(*
SPDX-FileCopyrightText: Â© 2026 Oleksandr Tiutyk <trofimich@gmail.com>
SPDX-License-Identifier: MIT
License: https://opensource.org/license/mit
*)

(*!
<summary>Represents a leaf automation component that performs cyclic output processing.</summary>
<description>
Invoked during the output phase of the component tree cycle to write physical outputs or command actuators.
</description>
*)

INTERFACE IOutputLeafAutomationComponent EXTENDS IChildAutomationComponent

(*!
<summary>Performs cyclic writing and processing of output data.</summary>
*)
METHOD ProcessOutput
END_METHOD

END_INTERFACE

(* stored: Version 1.1.0.1
   Itf IOutputLeafAutomationComponent: Id {9ff1eac2-7c3a-4e18-b5c3-83d36d605c6c}
   Method ProcessOutput: Id {5eb289e0-048e-4fb1-b4b5-450d3a21a673} *)
